// Mitsubishi GX Works2 project: CUARTO EJERCICIO   PLC: FX1S

PROGRAM MAIN
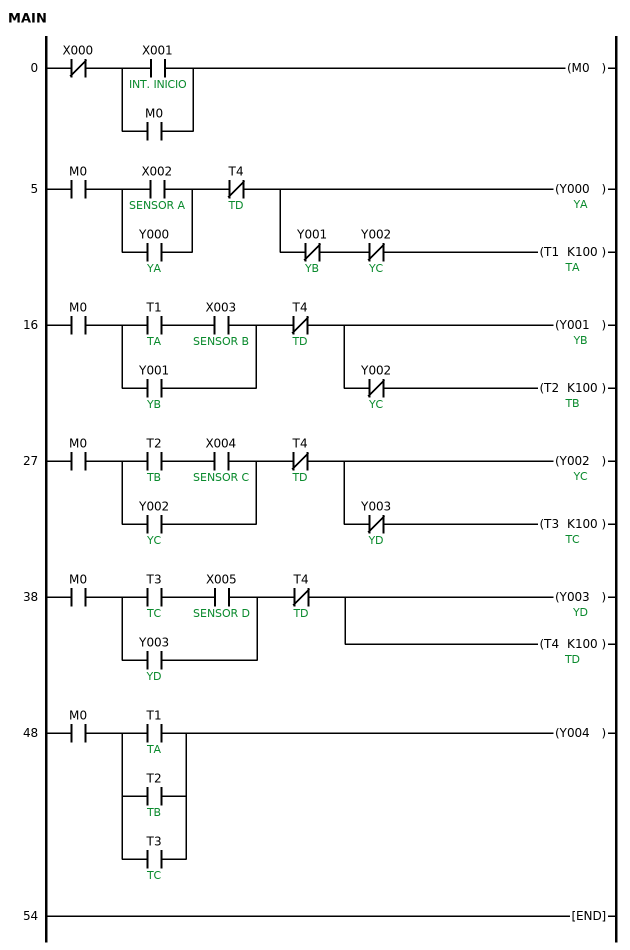
0     LDI     X000
      LD      X001  ; INT. INICIO
      OR      M0
      ANB
      OUT     M0
5     LD      M0
      LD      X002  ; SENSOR A
      OR      Y000  ; YA
      ANB
      ANI     T4  ; TD
      OUT     Y000  ; YA
      ANI     Y001  ; YB
      ANI     Y002  ; YC
      OUT     T1 K100  ; TA
16    LD      M0
      LD      T1  ; TA
      AND     X003  ; SENSOR B
      OR      Y001  ; YB
      ANB
      ANI     T4  ; TD
      OUT     Y001  ; YB
      ANI     Y002  ; YC
      OUT     T2 K100  ; TB
27    LD      M0
      LD      T2  ; TB
      AND     X004  ; SENSOR C
      OR      Y002  ; YC
      ANB
      ANI     T4  ; TD
      OUT     Y002  ; YC
      ANI     Y003  ; YD
      OUT     T3 K100  ; TC
38    LD      M0
      LD      T3  ; TC
      AND     X005  ; SENSOR D
      OR      Y003  ; YD
      ANB
      ANI     T4  ; TD
      OUT     Y003  ; YD
      OUT     T4 K100  ; TD
48    LD      M0
      LD      T1  ; TA
      OR      T2  ; TB
      OR      T3  ; TC
      ANB
      OUT     Y004
54    END
END_PROGRAM
